// TIA Portal project "Project6" (V14)

(* hardware
DEVICE "S7-1200 station_1"  S7-1200 Station
   slot 0: "Rack_0"  Rack  V1.0
   slot 1: "PLC_1"  CPU 1214C DC/DC/DC  6ES7 214-1AG40-0XB0  V4.1
DEVICE "HMI_1"  KTP400 Basic PN
   slot 0: "KTP400 Basic PN"  KTP400 Basic PN  6AV2 123-2DB03-0AX0  14.0.0.0
   slot 1: "HMI_RT_1"  KTP400 Basic PN  6AV2 123-2DB03-0AX0  14.0.0.0
   slot 5: "HMI_1.IE_CP_1"  PROFINET Interface  14.0.0.0
      slot 1: "PROFINET Interface_1"  PROFINET Interface
         slot 1: "Port_1"  Port
DEVICE "SINAMICS G_1"  Sinamics.Device
   slot 0: "	_0"  Rail
   slot 0: "CU 230 P"  G120P CU230P-2 PN  6SL3243-0BB30-1FA0  4.7.6
   slot 3: "PM240-2 IP20"  PM240-2 IP20  6SL3210-1PE11-8ULx  -
*)

// ===== PLC "PLC_1"  CPU 1214C DC/DC/DC =====
// protected blocks, not shown: "Denormalisation", "Main", "Normalisation", "Parameters", "Process_Data", "Simulation"

VAR_GLOBAL   // PLC tag table "Default tag table"
   "ZadanaBrzina" AT %MD0 : DInt;
   "TrenutnaBrzina" AT %MD2 : DInt;
   "TrenutnaStruja" AT %MD4 : DInt;
   "TrenutniNapon" AT %MD6 : DInt;
   "System_Byte" AT %MB1 : Byte;
   "FirstScan" AT %M1.0 : Bool;
   "DiagStatusUpdate" AT %M1.1 : Bool;
   "AlwaysTRUE" AT %M1.2 : Bool;
   "AlwaysFALSE" AT %M1.3 : Bool;
   "ON_OFF1" AT %M10.0 : Bool;
   "OFF2" AT %M10.1 : Bool;
   "OFF3" AT %M10.2 : Bool;
   "Ack" AT %M10.3 : Bool;
   "Dir_rev" AT %M10.4 : Bool;
   "Reset_SP" AT %M10.5 : Bool;
   "Inc_SP" AT %M10.6 : Bool;
   "Dec_SP" AT %M10.7 : Bool;
   "G120_1_PZD_I1" AT %IW256 : Word;
   "G120_1_PZD_I2" AT %IW258 : Word;
   "G120_1_PZD_I3" AT %IW260 : Word;
   "G120_1_PZD_I4" AT %IW262 : Word;
   "G120_1_PZD_I5" AT %IW264 : Word;
   "G120_1_PZD_I6" AT %IW266 : Word;
   "G120_1_PZD_Q1" AT %QW256 : Word;
   "G120_1_PZD_Q2" AT %QW258 : Word;
   "G120_1_PZD_Q3" AT %QW260 : Word;
   "G120_1_PZD_Q4" AT %QW262 : Word;
   "G120_1_PZD_Q5" AT %QW264 : Word;
   "G120_1_PZD_Q6" AT %QW266 : Word;
   "Clock_Byte" AT %MB0 : Byte;
   "Clock_10Hz" AT %M0.0 : Bool;
   "Clock_5Hz" AT %M0.1 : Bool;
   "Clock_2.5Hz" AT %M0.2 : Bool;
   "Clock_2Hz" AT %M0.3 : Bool;
   "Clock_1.25Hz" AT %M0.4 : Bool;
   "Clock_1Hz" AT %M0.5 : Bool;
   "Clock_0.625Hz" AT %M0.6 : Bool;
   "Clock_0.5Hz" AT %M0.7 : Bool;
   "System_Byte(1)" AT %MB1 : Byte;
END_VAR

DATA_BLOCK "idb_Process_Data"   // DB11
{ S7_Optimized_Access := 'TRUE' }
VERSION : 0.1
// stored: InstanceOfName Process_Data
"Process_Data"
BEGIN
END_DATA_BLOCK

DATA_BLOCK "idb_Parameters"   // DB20
{ S7_Optimized_Access := 'TRUE' }
VERSION : 0.1
// stored: InstanceOfName Parameters
"Parameters"
BEGIN
END_DATA_BLOCK

DATA_BLOCK "write_drive_parameters"   // DB100
TITLE = DB to send a write job to SINAMICS
{ S7_Optimized_Access := 'TRUE' }
VERSION : 2.0
   VAR
      record : Struct
         H_Reference : Byte;   // Head: Reference number
         H_Request_ID : Byte := 2;   // Head: Request ID: 1=read, 2=write
         H_Axis : Byte := 1;   // Head: Allways 1 for SINAMICS G120C
         H_Number_of_parameters : Byte := 2;   // Head: Number of parameters to transfer
         A_1_Attribute : Byte := 16#10;   // Address: 16#10 = parameter value
         A_1_Number_of_indices : Byte := 0;   // Address: Number of elements (0 to 234)
         A_1_Parameter_number : UInt := 1120;   // Address: Parameter number
         A_1_Index : UInt := 0;   // Address: Index number
         A_2_Attribute : Byte := 16#10;   // Address: 16#10 = parameter value
         A_2_Number_of_indices : Byte := 0;   // Address: Number of elements (0 to 234)
         A_2_Parameter_number : UInt := 1121;   // Address: Parameter number
         A_2_Index : UInt := 0;   // Address: Index number
         V_1_Format : Byte := 16#8;   // Value: Format of parameter value
         V_1_Number_of_index_values : Byte := 1;   // Value: Number of index values
         V_1_Value : Real := 10.0;   // Value: Parameter value
         V_2_Format : Byte := 16#8;   // Value: Format of parameter value
         V_2_Number_of_index_values : Byte := 1;   // Value: Number of index values
         V_2_Value : Real := 15.0;   // Value: Parameter value
      END_STRUCT;
   END_VAR
BEGIN
END_DATA_BLOCK

DATA_BLOCK "read_drive_parameters"   // DB101
TITLE = DB to send a read job to SINAMICS
{ S7_Optimized_Access := 'TRUE' }
VERSION : 2.0
   VAR
      record : Struct
         H_Reference : Byte;
         H_Request_ID : Byte := B#16#1;
         H_Axis : Byte := B#16#1;
         H_Number_of_parameters : Byte := B#16#3;
         A_1_Attribute : Byte := B#16#10;
         A_1_Number_of_indices : Byte;
         A_1_Parameter_number : Int := 1120;
         A_1_Index : Int;
         A_2_Attribute : Byte := B#16#10;
         A_2_Number_of_indices : Byte;
         A_2_Parameter_number : Int := 1121;
         A_2_Index : Int;
         A_3_Attribute : Byte := B#16#10;
         A_3_Number_of_indices : Byte := B#16#16;
         A_3_Parameter_number : Int := 945;
         A_3_Index : Int;
      END_STRUCT;
   END_VAR
BEGIN
END_DATA_BLOCK

DATA_BLOCK "answer_from_drive"   // DB103
TITLE = DB to receive from SINAMICS
{ S7_Optimized_Access := 'TRUE' }
VERSION : 0.1
   VAR
      record : Struct
         H_Reference : Byte;
         H_Response_ID : Byte;
         H_Axis : Byte;
         H_Number_of_parameters : Byte;
         V_1_Format : Byte;
         V_1_Number_of_index_valu : Byte;
         V_1_Value : Real;
         V_2_Format : Byte;
         V_2_Number_of_index_valu : Byte;
         V_2_Value : Real;
         V_3_Format : Byte;
         V_3_Number_of_index_valu : Byte;
         V_3_Value_00 : Word;
         V_3_Value_01 : Word;
         V_3_Value_02 : Word;
         V_3_Value_03 : Word;
         V_3_Value_04 : Word;
         V_3_Value_05 : Word;
         V_3_Value_06 : Word;
         V_3_Value_07 : Word;
         V_3_Value_08 : Word;
         V_3_Value_09 : Word;
         V_3_Value_10 : Word;
         V_3_Value_11 : Word;
         V_3_Value_12 : Word;
         V_3_Value_13 : Word;
         V_3_Value_14 : Word;
         V_3_Value_15 : Word;
      END_STRUCT;
   END_VAR
BEGIN
END_DATA_BLOCK

(* ===== HMI "HMI_RT_1" =====
system functions are stored by id; their names below are inferred from use
connection "HMI_Connection_1": ETHERNET, SMART_S7_1200_OMS

HMI tags "Default tag table"
   "Tag_ScreenNumber" : UInt, internal
   "ZadanaBrzina" : DInt = PLC ZadanaBrzina AT %MD0, 1 s
   "TrenutnaBrzina" : DInt = PLC TrenutnaBrzina AT %MD2, 1 s
   "TrenutniNapon" : DInt = PLC TrenutniNapon AT %MD6, 1 s
   "TrenutnaStruja" : DInt = PLC TrenutnaStruja AT %MD4, 1 s
   "zadana_brzina" : Real = PLC idb_Process_Data.setpoint AT %DB1.DBD0, 1 s
   "stvarna_brzina" : Real = PLC idb_Process_Data.actual_speed AT %DB1.DBD0, 1 s
   "stvarna_struja" : Real = PLC idb_Process_Data.actual_current AT %DB1.DBD0, 1 s
   "stvarni_moment" : Real = PLC idb_Process_Data.actual_torque AT %DB1.DBD0, 1 s
   "OFF2" : Bool = PLC OFF2 AT %M10.1, 1 s
   "ON_OFF1" : Bool = PLC ON_OFF1 AT %M10.0, 1 s
   "OFF3" : Bool = PLC OFF3 AT %M10.2, 1 s
   "Ack" : Bool = PLC Ack AT %M10.3, 1 s
   "Dir_rev" : Bool = PLC Dir_rev AT %M10.4, 1 s
   "Reset_SP" : Bool = PLC Reset_SP AT %M10.5, 1 s
   "Inc_SP" : Bool = PLC Inc_SP AT %M10.6, 1 s
   "Dec_SP" : Bool = PLC Dec_SP AT %M10.7, 1 s

